// TIA Portal V21 export
VAR_GLOBAL   // PLC tag table "K_Num"
END_VAR
VAR_GLOBAL CONSTANT   // user constants
   K_NumAnalogica : Int := 1;
   K_NumComunicazione : Int := 2;
   K_NumComunicazioneS7 : Int := 3;
   K_NumConsenso : Int := 4;
   K_NumDispositivoProfinet : Int := 5;
   K_NumMacchinaARicetta : Int := 6;
   K_NumMotore : Int := 2;
   K_NumNum : Int := 15;
   K_NumParatia : Int := 9;
   K_NumPid : Int := 10;
   K_NumPortata : Int := 11;
   K_NumSegnaliMacchina : Int := 12;
   K_NumSensore : Int := 13;
   K_NumSequenza : Int := 14;
   K_NumValvola : Int := 15;
   K_NumRicettaPerMacchina : Int := 1;
   K_NumZona : Int := 1;
   K_NumAdditivo : Int := 0;
END_VAR
